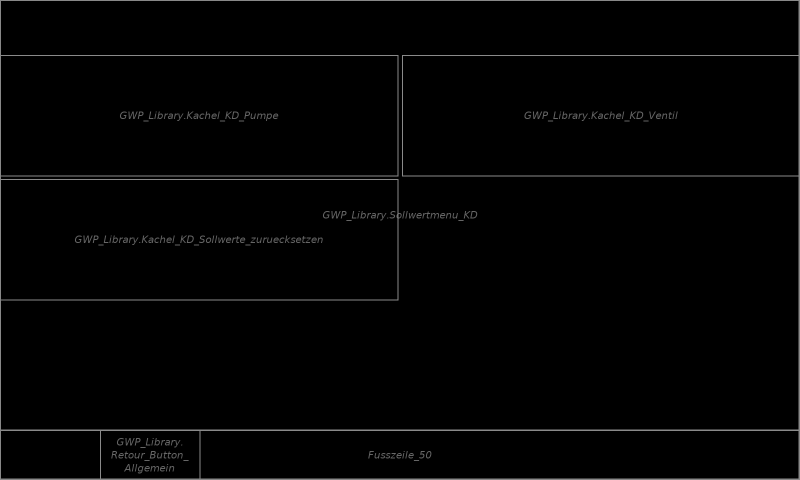
VISUALIZATION Sollwertmenu_KD  // 800x480
    Frame (0,0 800x430)
        shows GWP_Library.Sollwertmenu_KD()
    Frame (0,55 398x121)
        shows GWP_Library.Kachel_KD_Pumpe()
        OnMouseClick: change screen: KD_PU_Sollwerte
    Frame (402,55 398x121)
        shows GWP_Library.Kachel_KD_Ventil()
        OnMouseClick: change screen: KD_VTL_Sollwerte
    Frame (0,179 398x121)
        shows GWP_Library.Kachel_KD_Sollwerte_zuruecksetzen()
        OnMouseClick: change screen: KD_Sollwerte_zuruecksetzen
    Frame (0,430 800x50)
        shows Fusszeile_50()
    Frame (100,430 100x50)
        shows GWP_Library.Retour_Button_Allgemein()
END_VISUALIZATION

(* stored: Version 1.1.0.1, ProductVersion 3.1.4022.6
   Visu Sollwertmenu_KD: Id {81dbcd1c-6375-4208-a7dd-c9c426ba289a} *)
